Yaskawa INFORM job: GAUSSIANMOVING2.JBI

/JOB
//NAME GAUSSIANMOVING2
//POS
///NPOS 0,0,0,121,0,0
///TOOL 0
///POSTYPE ROBOT
///RECTAN
///RCONF 0,0,0,0,0,0,0,0,0,0,0,0,0,0,0,0,0,0,0,0,0,0,0,0
P00000=10.000,0.000,0.000,0.0000,0.0000,0.0000
///POSTYPE BASE
P00001=0272.90931211,0000.02795035,0483.09500000,0000.00000000,0000.00400000,0180.00000000,
P00002=0272.94917898,0000.03863264,0483.09500000,0000.00000000,0000.00400000,0180.00000000,
P00003=0273.00244531,0000.05290531,0483.09500000,0000.00000000,0000.00400000,0180.00000000,
P00004=0273.07290716,0000.07178551,0483.09500000,0000.00000000,0000.00400000,0180.00000000,
P00005=0273.16518895,0000.09651234,0483.09500000,0000.00000000,0000.00400000,0180.00000000,
P00006=0273.28484609,0000.12857437,0483.09500000,0000.00000000,0000.00400000,0180.00000000,
P00007=0273.43845693,0000.16973427,0483.09500000,0000.00000000,0000.00400000,0180.00000000,
P00008=0273.63369559,0000.22204831,0483.09500000,0000.00000000,0000.00400000,0180.00000000,
P00009=0273.87937592,0000.28787816,0483.09500000,0000.00000000,0000.00400000,0180.00000000,
P00010=0274.18545642,0000.36989218,0483.09500000,0000.00000000,0000.00400000,0180.00000000,
P00011=0274.56299520,0000.47105339,0483.09500000,0000.00000000,0000.00400000,0180.00000000,
P00012=0275.02404534,0000.59459141,0483.09500000,0000.00000000,0000.00400000,0180.00000000,
P00013=0275.58148185,0000.74395607,0483.09500000,0000.00000000,0000.00400000,0180.00000000,
P00014=0276.24875452,0000.92275124,0483.09500000,0000.00000000,0000.00400000,0180.00000000,
P00015=0277.03956409,0001.13464803,0483.09500000,0000.00000000,0000.00400000,0180.00000000,
P00016=0277.96746409,0001.38327808,0483.09500000,0000.00000000,0000.00400000,0180.00000000,
P00017=0279.04539542,0001.67210891,0483.09500000,0000.00000000,0000.00400000,0180.00000000,
P00018=0280.28516704,0002.00430472,0483.09500000,0000.00000000,0000.00400000,0180.00000000,
P00019=0281.69690130,0002.38257777,0483.09500000,0000.00000000,0000.00400000,0180.00000000,
P00020=0283.28846816,0002.80903683,0483.09500000,0000.00000000,0000.00400000,0180.00000000,
P00021=0285.06493658,0003.28504011,0483.09500000,0000.00000000,0000.00400000,0180.00000000,
P00022=0287.02807429,0003.81106127,0483.09500000,0000.00000000,0000.00400000,0180.00000000,
P00023=0289.17592807,0004.38657696,0483.09500000,0000.00000000,0000.00400000,0180.00000000,
P00024=0291.50251526,0005.00998411,0483.09500000,0000.00000000,0000.00400000,0180.00000000,
P00025=0293.99765355,0005.67855440,0483.09500000,0000.00000000,0000.00400000,0180.00000000,
P00026=0296.64695016,0006.38843129,0483.09500000,0000.00000000,0000.00400000,0180.00000000,
P00027=0299.43196312,0007.13467326,0483.09500000,0000.00000000,0000.00400000,0180.00000000,
P00028=0302.33053802,0007.91134407,0483.09500000,0000.00000000,0000.00400000,0180.00000000,
P00029=0305.31731303,0008.71164802,0483.09500000,0000.00000000,0000.00400000,0180.00000000,
P00030=0308.36437412,0009.52810558,0483.09500000,0000.00000000,0000.00400000,0180.00000000,
P00031=0311.44203305,0010.35276180,0483.09500000,0000.00000000,0000.00400000,0180.00000000,
P00032=0314.51969198,0011.17741803,0483.09500000,0000.00000000,0000.00400000,0180.00000000,
P00033=0317.56675308,0011.99387559,0483.09500000,0000.00000000,0000.00400000,0180.00000000,
P00034=0320.55352808,0012.79417954,0483.09500000,0000.00000000,0000.00400000,0180.00000000,
P00035=0323.45210299,0013.57085034,0483.09500000,0000.00000000,0000.00400000,0180.00000000,
P00036=0326.23711594,0014.31709232,0483.09500000,0000.00000000,0000.00400000,0180.00000000,
P00037=0328.88641255,0015.02696920,0483.09500000,0000.00000000,0000.00400000,0180.00000000,
P00038=0331.38155085,0015.69553949,0483.09500000,0000.00000000,0000.00400000,0180.00000000,
P00039=0333.70813803,0016.31894665,0483.09500000,0000.00000000,0000.00400000,0180.00000000,
P00040=0335.85599181,0016.89446234,0483.09500000,0000.00000000,0000.00400000,0180.00000000,
P00041=0337.81912952,0017.42048350,0483.09500000,0000.00000000,0000.00400000,0180.00000000,
P00042=0339.59559794,0017.89648678,0483.09500000,0000.00000000,0000.00400000,0180.00000000,
P00043=0341.18716480,0018.32294583,0483.09500000,0000.00000000,0000.00400000,0180.00000000,
P00044=0342.59889906,0018.70121889,0483.09500000,0000.00000000,0000.00400000,0180.00000000,
P00045=0343.83867068,0019.03341469,0483.09500000,0000.00000000,0000.00400000,0180.00000000,
P00046=0344.91660202,0019.32224553,0483.09500000,0000.00000000,0000.00400000,0180.00000000,
P00047=0345.84450201,0019.57087558,0483.09500000,0000.00000000,0000.00400000,0180.00000000,
P00048=0346.63531159,0019.78277237,0483.09500000,0000.00000000,0000.00400000,0180.00000000,
P00049=0347.30258425,0019.96156754,0483.09500000,0000.00000000,0000.00400000,0180.00000000,
P00050=0347.86002076,0020.11093220,0483.09500000,0000.00000000,0000.00400000,0180.00000000,
P00051=0348.32107090,0020.23447021,0483.09500000,0000.00000000,0000.00400000,0180.00000000,
P00052=0348.69860969,0020.33563143,0483.09500000,0000.00000000,0000.00400000,0180.00000000,
P00053=0349.00469018,0020.41764545,0483.09500000,0000.00000000,0000.00400000,0180.00000000,
P00054=0349.25037052,0020.48347529,0483.09500000,0000.00000000,0000.00400000,0180.00000000,
P00055=0349.44560917,0020.53578933,0483.09500000,0000.00000000,0000.00400000,0180.00000000,
P00056=0349.59922001,0020.57694924,0483.09500000,0000.00000000,0000.00400000,0180.00000000,
P00057=0349.71887715,0020.60901127,0483.09500000,0000.00000000,0000.00400000,0180.00000000,
P00058=0349.81115894,0020.63373810,0483.09500000,0000.00000000,0000.00400000,0180.00000000,
P00059=0349.88162079,0020.65261830,0483.09500000,0000.00000000,0000.00400000,0180.00000000,
P00060=0349.93488712,0020.66689097,0483.09500000,0000.00000000,0000.00400000,0180.00000000,
P00061=0132.67368789,-0000.02395035,0578.51100000,0000.00190000,-0000.28450000,0000.00000000
P00062=0132.63382102,-0000.03463264,0578.51100000,0000.00190000,-0000.28450000,0000.00000000
P00063=0132.58055469,-0000.04890531,0578.51100000,0000.00190000,-0000.28450000,0000.00000000
P00064=0132.51009284,-0000.06778551,0578.51100000,0000.00190000,-0000.28450000,0000.00000000
P00065=0132.41781105,-0000.09251234,0578.51100000,0000.00190000,-0000.28450000,0000.00000000
P00066=0132.29815391,-0000.12457437,0578.51100000,0000.00190000,-0000.28450000,0000.00000000
P00067=0132.14454307,-0000.16573427,0578.51100000,0000.00190000,-0000.28450000,0000.00000000
P00068=0131.94930441,-0000.21804831,0578.51100000,0000.00190000,-0000.28450000,0000.00000000
P00069=0131.70362408,-0000.28387816,0578.51100000,0000.00190000,-0000.28450000,0000.00000000
P00070=0131.39754358,-0000.36589218,0578.51100000,0000.00190000,-0000.28450000,0000.00000000
P00071=0131.02000480,-0000.46705339,0578.51100000,0000.00190000,-0000.28450000,0000.00000000
P00072=0130.55895466,-0000.59059141,0578.51100000,0000.00190000,-0000.28450000,0000.00000000
P00073=0130.00151815,-0000.73995607,0578.51100000,0000.00190000,-0000.28450000,0000.00000000
P00074=0129.33424548,-0000.91875124,0578.51100000,0000.00190000,-0000.28450000,0000.00000000
P00075=0128.54343591,-0001.13064803,0578.51100000,0000.00190000,-0000.28450000,0000.00000000
P00076=0127.61553591,-0001.37927808,0578.51100000,0000.00190000,-0000.28450000,0000.00000000
P00077=0126.53760458,-0001.66810891,0578.51100000,0000.00190000,-0000.28450000,0000.00000000
P00078=0125.29783296,-0002.00030472,0578.51100000,0000.00190000,-0000.28450000,0000.00000000
P00079=0123.88609870,-0002.37857777,0578.51100000,0000.00190000,-0000.28450000,0000.00000000
P00080=0122.29453184,-0002.80503683,0578.51100000,0000.00190000,-0000.28450000,0000.00000000
P00081=0120.51806342,-0003.28104011,0578.51100000,0000.00190000,-0000.28450000,0000.00000000
P00082=0118.55492571,-0003.80706127,0578.51100000,0000.00190000,-0000.28450000,0000.00000000
P00083=0116.40707193,-0004.38257696,0578.51100000,0000.00190000,-0000.28450000,0000.00000000
P00084=0114.08048474,-0005.00598411,0578.51100000,0000.00190000,-0000.28450000,0000.00000000
P00085=0111.58534645,-0005.67455440,0578.51100000,0000.00190000,-0000.28450000,0000.00000000
P00086=0108.93604984,-0006.38443129,0578.51100000,0000.00190000,-0000.28450000,0000.00000000
P00087=0106.15103688,-0007.13067326,0578.51100000,0000.00190000,-0000.28450000,0000.00000000
P00088=0103.25246198,-0007.90734407,0578.51100000,0000.00190000,-0000.28450000,0000.00000000
P00089=0100.26568697,-0008.70764802,0578.51100000,0000.00190000,-0000.28450000,0000.00000000
P00090=0097.21862588,-0009.52410558,0578.51100000,0000.00190000,-0000.28450000,0000.00000000
P00091=0094.14096695,-0010.34876180,0578.51100000,0000.00190000,-0000.28450000,0000.00000000
P00092=0091.06330802,-0011.17341803,0578.51100000,0000.00190000,-0000.28450000,0000.00000000
P00093=0088.01624692,-0011.98987559,0578.51100000,0000.00190000,-0000.28450000,0000.00000000
P00094=0085.02947192,-0012.79017954,0578.51100000,0000.00190000,-0000.28450000,0000.00000000
P00095=0082.13089701,-0013.56685034,0578.51100000,0000.00190000,-0000.28450000,0000.00000000
P00096=0079.34588406,-0014.31309232,0578.51100000,0000.00190000,-0000.28450000,0000.00000000
P00097=0076.69658745,-0015.02296920,0578.51100000,0000.00190000,-0000.28450000,0000.00000000
P00098=0074.20144915,-0015.69153949,0578.51100000,0000.00190000,-0000.28450000,0000.00000000
P00099=0071.87486197,-0016.31494665,0578.51100000,0000.00190000,-0000.28450000,0000.00000000
P00100=0069.72700819,-0016.89046234,0578.51100000,0000.00190000,-0000.28450000,0000.00000000
P00101=0067.76387048,-0017.41648350,0578.51100000,0000.00190000,-0000.28450000,0000.00000000
P00102=0065.98740206,-0017.89248678,0578.51100000,0000.00190000,-0000.28450000,0000.00000000
P00103=0064.39583520,-0018.31894583,0578.51100000,0000.00190000,-0000.28450000,0000.00000000
P00104=0062.98410094,-0018.69721889,0578.51100000,0000.00190000,-0000.28450000,0000.00000000
P00105=0061.74432932,-0019.02941469,0578.51100000,0000.00190000,-0000.28450000,0000.00000000
P00106=0060.66639798,-0019.31824553,0578.51100000,0000.00190000,-0000.28450000,0000.00000000
P00107=0059.73849799,-0019.56687558,0578.51100000,0000.00190000,-0000.28450000,0000.00000000
P00108=0058.94768841,-0019.77877237,0578.51100000,0000.00190000,-0000.28450000,0000.00000000
P00109=0058.28041575,-0019.95756754,0578.51100000,0000.00190000,-0000.28450000,0000.00000000
P00110=0057.72297924,-0020.10693220,0578.51100000,0000.00190000,-0000.28450000,0000.00000000
P00111=0057.26192910,-0020.23047021,0578.51100000,0000.00190000,-0000.28450000,0000.00000000
P00112=0056.88439031,-0020.33163143,0578.51100000,0000.00190000,-0000.28450000,0000.00000000
P00113=0056.57830982,-0020.41364545,0578.51100000,0000.00190000,-0000.28450000,0000.00000000
P00114=0056.33262948,-0020.47947529,0578.51100000,0000.00190000,-0000.28450000,0000.00000000
P00115=0056.13739083,-0020.53178933,0578.51100000,0000.00190000,-0000.28450000,0000.00000000
P00116=0055.98377999,-0020.57294924,0578.51100000,0000.00190000,-0000.28450000,0000.00000000
P00117=0055.86412285,-0020.60501127,0578.51100000,0000.00190000,-0000.28450000,0000.00000000
P00118=0055.77184106,-0020.62973810,0578.51100000,0000.00190000,-0000.28450000,0000.00000000
P00119=0055.70137921,-0020.64861830,0578.51100000,0000.00190000,-0000.28450000,0000.00000000
P00120=0055.64811288,-0020.66289097,0578.51100000,0000.00190000,-0000.28450000,0000.00000000
//INST
///DATE 2017/03/31 08:11
///COMM PLAYINGTWOROBOTS
///ATTR SC,RW
///GROUP1 RB1
///GROUP2 RB2
NOP
MOVL P00001 V=0002.5795763  +MOVL P00061 V=0002.5795763
MOVL P00002 V=0003.4465852  +MOVL P00062 V=0003.4465852
MOVL P00003 V=0004.5592174  +MOVL P00063 V=0004.5592174
MOVL P00004 V=0005.9710711  +MOVL P00064 V=0005.9710711
MOVL P00005 V=0007.7423865  +MOVL P00065 V=0007.7423865
MOVL P00006 V=0009.9393530  +MOVL P00066 V=0009.9393530
MOVL P00007 V=0012.6328705  +MOVL P00067 V=0012.6328705
MOVL P00008 V=0015.8966875  +MOVL P00068 V=0015.8966875
MOVL P00009 V=0019.8048652  +MOVL P00069 V=0019.8048652
MOVL P00010 V=0024.4285569  +MOVL P00070 V=0024.4285569
MOVL P00011 V=0029.8321393  +MOVL P00071 V=0029.8321393
MOVL P00012 V=0036.0687965  +MOVL P00072 V=0036.0687965
MOVL P00013 V=0043.1757182  +MOVL P00073 V=0043.1757182
MOVL P00014 V=0051.1691447  +MOVL P00074 V=0051.1691447
MOVL P00015 V=0060.0395478  +MOVL P00075 V=0060.0395478
MOVL P00016 V=0069.7472898  +MOVL P00076 V=0069.7472898
MOVL P00017 V=0080.2191268  +MOVL P00077 V=0080.2191268
MOVL P00018 V=0091.3459282  +MOVL P00078 V=0091.3459282
MOVL P00019 V=0102.9819536  +MOVL P00079 V=0102.9819536
MOVL P00020 V=0114.9459649  +MOVL P00080 V=0114.9459649
MOVL P00021 V=0127.0243571  +MOVL P00081 V=0127.0243571
MOVL P00022 V=0138.9763662  +MOVL P00082 V=0138.9763662
MOVL P00023 V=0150.5412682  +MOVL P00083 V=0150.5412682
MOVL P00024 V=0161.4473276  +MOVL P00084 V=0161.4473276
MOVL P00025 V=0171.4221049  +MOVL P00085 V=0171.4221049
MOVL P00026 V=0180.2035983  +MOVL P00086 V=0180.2035983
MOVL P00027 V=0187.5515971  +MOVL P00087 V=0187.5515971
MOVL P00028 V=0193.2585637  +MOVL P00088 V=0193.2585637
MOVL P00029 V=0197.1593608  +MOVL P00089 V=0197.1593608
MOVL P00030 V=0199.1391864  +MOVL P00090 V=0199.1391864
MOVL P00031 V=0199.1391864  +MOVL P00091 V=0199.1391864
MOVL P00032 V=0197.1593608  +MOVL P00092 V=0197.1593608
MOVL P00033 V=0193.2585637  +MOVL P00093 V=0193.2585637
MOVL P00034 V=0187.5515971  +MOVL P00094 V=0187.5515971
MOVL P00035 V=0180.2035983  +MOVL P00095 V=0180.2035983
MOVL P00036 V=0171.4221049  +MOVL P00096 V=0171.4221049
MOVL P00037 V=0161.4473276  +MOVL P00097 V=0161.4473276
MOVL P00038 V=0150.5412682  +MOVL P00098 V=0150.5412682
MOVL P00039 V=0138.9763662  +MOVL P00099 V=0138.9763662
MOVL P00040 V=0127.0243571  +MOVL P00100 V=0127.0243571
MOVL P00041 V=0114.9459649  +MOVL P00101 V=0114.9459649
MOVL P00042 V=0102.9819536  +MOVL P00102 V=0102.9819536
MOVL P00043 V=0091.3459282  +MOVL P00103 V=0091.3459282
MOVL P00044 V=0080.2191268  +MOVL P00104 V=0080.2191268
MOVL P00045 V=0069.7472898  +MOVL P00105 V=0069.7472898
MOVL P00046 V=0060.0395478  +MOVL P00106 V=0060.0395478
MOVL P00047 V=0051.1691447  +MOVL P00107 V=0051.1691447
MOVL P00048 V=0043.1757182  +MOVL P00108 V=0043.1757182
MOVL P00049 V=0036.0687965  +MOVL P00109 V=0036.0687965
MOVL P00050 V=0029.8321393  +MOVL P00110 V=0029.8321393
MOVL P00051 V=0024.4285569  +MOVL P00111 V=0024.4285569
MOVL P00052 V=0019.8048652  +MOVL P00112 V=0019.8048652
MOVL P00053 V=0015.8966875  +MOVL P00113 V=0015.8966875
MOVL P00054 V=0012.6328705  +MOVL P00114 V=0012.6328705
MOVL P00055 V=0009.9393530  +MOVL P00115 V=0009.9393530
MOVL P00056 V=0007.7423865  +MOVL P00116 V=0007.7423865
MOVL P00057 V=0005.9710711  +MOVL P00117 V=0005.9710711
MOVL P00058 V=0004.5592174  +MOVL P00118 V=0004.5592174
MOVL P00059 V=0003.4465852  +MOVL P00119 V=0003.4465852
MOVL P00060 V=0003.4465852  +MOVL P00120 V=0003.4465852
END
